INTERFACE ITaskState

METHOD Cyclic
END_METHOD

METHOD Inihibits : BOOL
VAR_INPUT
END_VAR
END_METHOD

METHOD newCommandState : BOOL
VAR_INPUT
	newTaskState : ENUM;
END_VAR
END_METHOD

PROPERTY newTaskCommand : BOOL
GET
END_GET
END_PROPERTY

METHOD stateErrored : BOOL
VAR_INPUT
END_VAR
END_METHOD

METHOD stateFinished : BOOL
VAR_INPUT
END_VAR
END_METHOD

METHOD StateMachine : BOOL
VAR_INPUT
END_VAR
END_METHOD

{attribute 'monitoring' := 'call'}
PROPERTY taskReady : Bool
GET
END_GET
SET
END_SET
END_PROPERTY

{attribute 'monitoring' := 'call'}
PROPERTY taskState : ENUM
GET
END_GET
END_PROPERTY

METHOD UpdateState : BOOL
VAR_INPUT
END_VAR
END_METHOD

END_INTERFACE

(* stored: Version 1.1.0.1
   Itf ITaskState: Id {c414fd66-a244-4c63-a9ca-a3748ab93237}
   Method Cyclic: Id {df7848e1-6796-42e6-952c-938fef13bd38}
   Method Inihibits: Id {e83ce640-e6f2-45e5-949b-c526c3174821}
   Method newCommandState: Id {8fecb899-e712-4c2b-84b8-942531440e9a}
   Property newTaskCommand: Id {6790c3f8-5fb9-444d-9490-9a806808eff2}
   Get Get: Id {4a221e21-683f-4623-87f8-f23f402dd6ee}
   Method stateErrored: Id {1a290f15-f898-411f-a486-cdd0d8c7bba2}
   Method stateFinished: Id {cd0661c2-8f19-4da1-9ffb-aae73db39d56}
   Method StateMachine: Id {8686b074-f9b6-4442-b1e6-0de110cfebc5}
   Property taskReady: Id {bd8a546f-5904-4116-aebd-80d37e3d8855}
   Get Get: Id {ee69b286-51fd-41c8-ba24-ab7d84cccfed}
   Set Set: Id {ec0be226-c73b-41e3-8440-7511474e4879}
   Property taskState: Id {17386119-9411-446c-9999-0b14544f8dcf}
   Get Get: Id {965a4deb-c78d-498e-bc57-5a24822c86ee}
   Method UpdateState: Id {bae77c85-768e-452a-8e93-0534a052dc9c} *)
